// TIA Portal project "BT_MOVEMENT_lesson14" (V19)

(* hardware
DEVICE "PC-System_1"  SIMATIC PC station
   slot 0: "SIMATIC PC station"  Rail  SIMATIC PC-Station  V1.0
      slot 125: "Stationmanager"  Station_Manager  V6.0.4
   slot 1: "HMI_RT_1"  WinCC RT Advanced  6AV2 104-0xxxx-xxxx  17.0.0.0
      slot 33792: "Computer interface"  Host interface
   slot 2: "IE general_1"  IE General  IE_CP  V8.2.0
      slot 1: "PROFINET interface"  IEGeneral.Interface.8.2.0
DEVICE "S7-1200 station_1"  S7-1200 Station
   slot 0: "Rack_0"  S7-1200 Rack  Rack  V1.0
   slot 1: "PLC_1"  CPU 1212C AC/DC/Rly  6ES7 212-1BE40-0XB0  V4.6
*)

// ===== PLC "PLC_1"  CPU 1212C AC/DC/Rly =====

VAR_GLOBAL   // PLC tag table "Default tag table"
   "Tag_1" AT %M25.0 : Bool;
   "Tag_2" AT %M21.1 : Bool;
END_VAR

VAR_GLOBAL   // PLC tag table "MOVEMENT"
   "BUTTON_ON" AT %M0.0 : Bool;
   "BUTTON_OFF" AT %M0.1 : Bool;
   "CONVEYOR" AT %Q0.0 : Bool;
   "Product_Counter" AT %MW10 : Int;
   "SENSOR" AT %M20.0 : Bool;
END_VAR

// folder: System blocks/Program resources

DATA_BLOCK "Timer_Simulation_Movement"   // DB1
{ S7_Optimized_Access := 'TRUE' }
AUTHOR : Simatic
FAMILY : IEC
NAME : IEC_TMR
VERSION : 1.0
// stored: InstanceOfName IEC_TIMER
"IEC_TIMER"
BEGIN
END_DATA_BLOCK

// folder: (top level)

ORGANIZATION_BLOCK "Main"   // OB1, LAD, ProgramCycle
TITLE = "Main Program Sweep (Cycle)"
{ S7_Optimized_Access := 'TRUE' }
VERSION : 0.1
   VAR_INPUT
      Initial_Call : Bool;   // Initial call of this OB
      Remanence : Bool;   // =True, if remanent data are available
   END_VAR
   VAR_TEMP   // added for the SCL form of the ladder/FBD networks
      _w1 : Bool;
   END_VAR
BEGIN

REGION Network 1: Turn ON/OFF conveyor
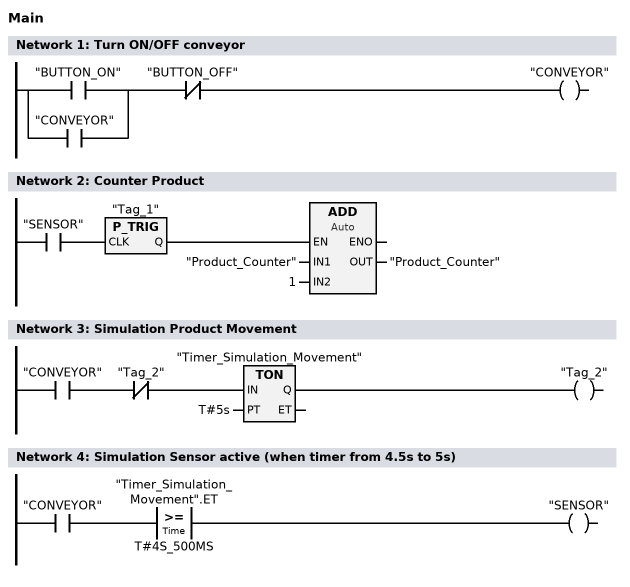
   RUNG wire#powerrail
      Contact( "BUTTON_ON" )
      wire#w1
      I_Contact( "BUTTON_OFF" )
      Coil( "CONVEYOR" )
   END_RUNG
   RUNG wire#powerrail
      Contact( "CONVEYOR" )
   END_RUNG wire#w1
   // the same network as SCL:
   "CONVEYOR" := ("BUTTON_ON" OR "CONVEYOR") AND NOT "BUTTON_OFF";
END_REGION

REGION Network 2: Counter Product
   RUNG wire#powerrail
      Contact( "SENSOR" )
      P_Trig( "Tag_1" )
      Add(in1 := "Product_Counter", in2 := 1, out => "Product_Counter")
   END_RUNG
   // the same network as SCL:
   #_w1 := "SENSOR" AND NOT "Tag_1";   // rising edge
   "Tag_1" := "SENSOR";
   IF #_w1 THEN "Product_Counter" := "Product_Counter" + 1; END_IF;
END_REGION

REGION Network 3: Simulation Product Movement
   "Timer_Simulation_Movement".TON(IN := "CONVEYOR" AND NOT "Tag_2", PT := T#5s);
   "Tag_2" := "Timer_Simulation_Movement".Q;
END_REGION

REGION Network 4: Simulation Sensor active (when timer from 4.5s to 5s)
   RUNG wire#powerrail
      Contact( "CONVEYOR" )
      { S7_Templates := "SrcType := Time" } GE_Contact(in1 := "Timer_Simulation_Movement".ET, in2 := T#4S_500MS)
      Coil( "SENSOR" )
   END_RUNG
   // the same network as SCL:
   "SENSOR" := "CONVEYOR" AND ("Timer_Simulation_Movement".ET >= T#4S_500MS);
END_REGION
END_ORGANIZATION_BLOCK

(* ===== HMI "HMI_RT_1" =====
system functions are stored by id; their names below are inferred from use
connection "HMI_Connection_1": ETHERNET, S7_1200_OMS

HMI tags "Default tag table"
   "Timer_Simulation_Movement_ET" : Time = PLC Timer_Simulation_Movement.ET, 100 ms
   "CONVEYOR" : Bool = PLC CONVEYOR AT %Q0.0, 100 ms
   "Product_Counter" : Int = PLC Product_Counter AT %MW10, 100 ms
   "SENSOR" : Bool = PLC SENSOR AT %M20.0, 100 ms
   "BUTTON_ON" : Bool = PLC BUTTON_ON AT %M0.0, 100 ms
   "BUTTON_OFF" : Bool = PLC BUTTON_OFF AT %M0.1, 100 ms

screen "Screen_1" 1024x768
   SymbolLibrary "Symbol library_1" at 81,342 size 388x54
      Appearance <- "CONVEYOR"
   SymbolLibrary "Symbol library_2" at 323,342 size 388x54
      Appearance <- "CONVEYOR"
      on Press: SetBit("BUTTON_ON")
      on Release: ResetBit("BUTTON_ON")
   SymbolLibrary "Symbol library_3" at 650,172 size 41x62
      Appearance <- "SENSOR"
   SymbolLibrary "Symbol library_4" at 142,294 size 34x70
      HorizontalMovement <- "Timer_Simulation_Movement_ET"
   Button "Button_1" at 783,294 size 96x32; TextOff 'ON'
      Appearance <- "CONVEYOR"
      on Press: SetBit("BUTTON_ON")
      on Release: ResetBit("BUTTON_ON")
   Button "Button_2" at 785,347 size 96x32; TextOff 'OFF'
      Appearance <- "CONVEYOR"
      on Press: SetBit("BUTTON_OFF")
      on Release: ResetBit("BUTTON_OFF")
   SymbolLibrary "Symbol library_5" at 139,417 size 74x61
      Appearance <- "CONVEYOR"
   IOField "I/O field_1" at 626,134 size 84x32; FormatPattern 99999
      ProcessValue <- "Product_Counter"
   TextField "Text field_1" at 718,138 size 39x22; Text '[SP]'
*)